(* CoDeSys 2.3 export: NETVARTELEGRAMM_UDP.EXP *)

(* Data type *)
TYPE NetVarTelegramm_Udp:
STRUCT
	Header		: NetVarTlgHeader_Udp;
	pData		: ARRAY[0..256] OF BYTE;
END_STRUCT
END_TYPE
